{attribute 'linkalways'} 
{attribute 'no_explicit_call' := 'This FB is a CLASS and must be accessed using methods or properties'}
{attribute 'enable_dynamic_creation'}
FUNCTION_BLOCK Node_ContainerType_Vector_REAL EXTENDS Node
VAR
    out : _GUID;
END_VAR

METHOD PUBLIC  Clone : I_Node
VAR
	pNode : POINTER TO Node_ContainerType_Vector_REAL;
END_VAR
pNode := __NEW(Node_ContainerType_Vector_REAL);
Clone := pNode^;
END_METHOD

METHOD FB_init : BOOL
VAR_INPUT
	bInitRetains : BOOL; // if TRUE, the retain variables are initialized (warm start / cold start)
	bInCopyCode : BOOL;  // if TRUE, the instance afterwards gets moved into the copy code (online change)
END_VAR
AddOutput('out', out);
END_METHOD

METHOD PROTECTED OnExecute
out.Value := ContainerType_Vector_REAL;
END_METHOD

END_FUNCTION_BLOCK

(* stored: Version 1.1.0.1, ProductVersion 3.1.4026.17
   POU Node_ContainerType_Vector_REAL: Id {61b30199-73fc-0b58-0658-23ba0e51b64f}, SpecialFunc None
   Folder Constructor: Id {9218ea7f-3859-0ae0-3c45-e8d3abab39a7}
   Method Clone: Id {317d3a01-603b-0fdb-2faf-66d6d06cf461}
   Method FB_init: Id {121d36f7-76ce-0bad-3b2b-31e2012d8d18}
   Method OnExecute: Id {bcebfa5f-d95b-071c-1d9f-059fb11087a4} *)
